// TIA Portal V17 export
// export: Created 2022-07-06T14:39:44.2676002Z, ExportSetting WithDefaults, DisplayName Totally Integrated Automation Portal, DisplayVersion V17 Update 4, DisplayName TIA Portal Openness, DisplayVersion V17 Update 4, DisplayName TIA Portal Version Control Interface, DisplayVersion V17, DisplayName STEP 7 Professional, DisplayVersion V17 Update 4, DisplayName STEP 7 CFC, DisplayVersion V17, DisplayName STEP 7 Safety, DisplayVersion V17, DisplayName WinCC Advanced, DisplayVersion V17 Update 4
DATA_BLOCK "HDB_STR"   // DB4300
{ S7_Optimized_Access := 'FALSE' }
NAME : DEV
VERSION : 0.1
// stored: AutoNumber false, DBAccessibleFromOPCUA true, IsOnlyStoredInLoadMemory false, IsWriteProtectedInAS false
   VAR RETAIN
      Cmd_ResetOsKnf1Top : Bool := FALSE;   // Knife 1 ss reset mileage
      Cmd_ResetOsKnf1Bot : Bool := FALSE;   // Knife 2 ss reset mileage
      Cmd_ResetOsSchp1 : Bool := FALSE;   // Knife 1 bs reset mileage
      Cmd_ResetOsKnf2Top : Bool := FALSE;   // Knife 1 ss reset mileage
      Cmd_ResetOsKnf2Bot : Bool := FALSE;   // Knife 2 ss reset mileage
      Cmd_ResetOsSchp2 : Bool := FALSE;   // Knife 1 bs reset mileage
      Cmd_ResetDsKnf1Top : Bool := FALSE;   // Knife 1 ss reset mileage
      Cmd_ResetDsKnf1Bot : Bool := FALSE;   // Knife 2 ss reset mileage
      Cmd_ResetDsSchp1 : Bool := FALSE;   // Knife 1 bs reset mileage
      Cmd_ResetDsKnf2Top : Bool := FALSE;   // Knife 1 ss reset mileage
      Cmd_ResetDsKnf2Bot : Bool := FALSE;   // Knife 2 ss reset mileage
      Cmd_ResetDsSchp2 : Bool := FALSE;   // Knife 1 bs reset mileage
      Cmd_FrcNotchInPos : Bool := FALSE;   // Notch in position
      Cmd_AutoRestart : Bool := FALSE;   // Line automatic start
      Cmd_StopRqst : Bool := FALSE;   // Line stop request
      Cmd_KnifeChngOsKnf1 : Bool := FALSE;   // Knife change operator Side Knife 1 request / Knife change BAL Side Knife 1 request
      Cmd_KnifeChngOsKnf2 : Bool := FALSE;   // Knife change operator Side Knife 2 request / Knife change BAL Side Knife 2 request
      Cmd_KnifeChngDsKnf1 : Bool := FALSE;   // Knife change drive Side Knife 1 request / Knife change Street Side Knife 1 request
      Cmd_KnifeChngDsKnf2 : Bool := FALSE;   // Knife change drive Side Knife 2 request / Knife change Street Side Knife 2 request
      Cmd_Spare23 { ExternalAccessible := 'False'; ExternalVisible := 'False'; ExternalWritable := 'False'} : Bool;
      Cmd_Spare24 { ExternalAccessible := 'False'; ExternalVisible := 'False'; ExternalWritable := 'False'} : Bool;
      Cmd_Spare25 { ExternalAccessible := 'False'; ExternalVisible := 'False'; ExternalWritable := 'False'} : Bool;
      Cmd_Spare26 { ExternalAccessible := 'False'; ExternalVisible := 'False'; ExternalWritable := 'False'} : Bool;
      Cmd_Spare27 { ExternalAccessible := 'False'; ExternalVisible := 'False'; ExternalWritable := 'False'} : Bool;
      Cmd_Spare31 { ExternalAccessible := 'False'; ExternalVisible := 'False'; ExternalWritable := 'False'} : Bool;
      Cmd_Spare32 { ExternalAccessible := 'False'; ExternalVisible := 'False'; ExternalWritable := 'False'} : Bool;
      Cmd_Spare33 { ExternalAccessible := 'False'; ExternalVisible := 'False'; ExternalWritable := 'False'} : Bool;
      Cmd_Spare34 { ExternalAccessible := 'False'; ExternalVisible := 'False'; ExternalWritable := 'False'} : Bool;
      Cmd_Spare35 { ExternalAccessible := 'False'; ExternalVisible := 'False'; ExternalWritable := 'False'} : Bool;
      Cmd_Spare36 { ExternalAccessible := 'False'; ExternalVisible := 'False'; ExternalWritable := 'False'} : Bool;
      Cmd_Spare37 { ExternalAccessible := 'False'; ExternalVisible := 'False'; ExternalWritable := 'False'} : Bool;
      Stat_NotchInPos : DInt := 4;   // Status notch in position
      Stat_AutoRestart : DInt := 6;   // Status Line automatic start
      Stat_StopRqst : DInt := 4;   // Status Line stop request
      Stat_KnifeChngOsKnf1 : DInt := 4;   // Status Knife change operator side Knife 1 request / Status Knife change BAL side Knife 1 request
      Stat_KnifeChngOsKnf2 : DInt := 1;   // Status Knife change operator side Knife 2 request / Status Knife change BAL side Knife 2 request
      Stat_KnifeChngDsKnf1 : DInt := 1;   // Status Knife change drive side Knife 1 request / Status Knife change Street side Knife 1 request
      Stat_KnifeChngDsKnf2 : DInt := 4;   // Status Knife change drive side Knife 2 request / Status Knife change Street side Knife 2 request
      Stat_Spare1 { ExternalAccessible := 'False'; ExternalVisible := 'False'; ExternalWritable := 'False'} : DInt;
      Stat_Spare2 { ExternalAccessible := 'False'; ExternalVisible := 'False'; ExternalWritable := 'False'} : DInt;
      Stat_Spare3 { ExternalAccessible := 'False'; ExternalVisible := 'False'; ExternalWritable := 'False'} : DInt;
      Stat_Spare4 { ExternalAccessible := 'False'; ExternalVisible := 'False'; ExternalWritable := 'False'} : DInt;
      Stat_Spare5 { ExternalAccessible := 'False'; ExternalVisible := 'False'; ExternalWritable := 'False'} : DInt;
      Chopper_Overspeed { S7_SetPoint := 'True'} : Real := 1.0;   // Chopper overspeed [%]
      MileageOsKnf1Top { S7_SetPoint := 'True'} : Real := 29.0;   // Mileage of knife 1 top OS / Mileage of knife 1 top Ss
      MileageOsKnf1Bot { S7_SetPoint := 'True'} : Real;   // Mileage of knife 1 bottom OS
      MileageOsSchp1 { S7_SetPoint := 'True'} : Real := 29.54701;   // Mileage of scrap chopper knife 1 OS / Mileage of scrap chopper knife 1 Ss
      MileageOsKnf2Top { S7_SetPoint := 'True'} : Real := 29.54701;   // Mileage of knife 2 top OS / Mileage of knife 1 top Ss
      MileageOsKnf2Bot { S7_SetPoint := 'True'} : Real;   // Mileage of knife 2 bottom OS
      MileageOsSchp2 { S7_SetPoint := 'True'} : Real := 18.93003;   // Mileage of scrap chopper knife 2 OS / Mileage of scrap chopper knife 2 Ss
      MileageDsKnf1Top { S7_SetPoint := 'True'} : Real := 29.54701;   // Mileage of knife 1 top DS / Mileage of knife 1 top Ss
      MileageDsKnf1Bot { S7_SetPoint := 'True'} : Real;   // Mileage of knife 1 bottom DS
      MileageDsSchp1 { S7_SetPoint := 'True'} : Real := 29.54701;   // Mileage of scrap chopper knife 1 DS / Mileage of scrap chopper knife 1 Ss
      MileageDsKnf2Top { S7_SetPoint := 'True'} : Real := 29.54701;   // Mileage of knife 2 top DS / Mileage of knife 1 top Ss
      MileageDsKnf2Bot { S7_SetPoint := 'True'} : Real;   // Mileage of knife 2 bottom DS
      MileageDsSchp2 { S7_SetPoint := 'True'} : Real := 18.93003;   // Mileage of scrap chopper knife 2 DS / Mileage of scrap chopper knife 2 Ss
      SetpOsGapKnf1 { S7_SetPoint := 'True'} : "SplSetpCtrl";   // Setpoint OS gap knife 1
      SetpOsOvlKnf1 { S7_SetPoint := 'True'} : "SplSetpCtrl";   // Setpoint OS overlap knife 1
      SetpOsSchp1 { S7_SetPoint := 'True'} : "SplSetpCtrl";   // Setpoint OS gap scrap chopper 1
      SetpOsGapKnf2 { S7_SetPoint := 'True'} : "SplSetpCtrl";   // Setpoint OS gap knife 2
      SetpOsOvlKnf2 { S7_SetPoint := 'True'} : "SplSetpCtrl";   // Setpoint OS overlap knife 2
      SetpOsSchp2 { S7_SetPoint := 'True'} : "SplSetpCtrl";   // Setpoint OS gap scrap chopper 2
      SetpDsGapKnf1 { S7_SetPoint := 'True'} : "SplSetpCtrl";   // Setpoint DS gap knife 1
      SetpDsOvlKnf1 { S7_SetPoint := 'True'} : "SplSetpCtrl";   // Setpoint DS overlap knife 1
      SetpDsSchp1 { S7_SetPoint := 'True'} : "SplSetpCtrl";   // Setpoint DS gap scrap chopper 1
      SetpDsGapKnf2 { S7_SetPoint := 'True'} : "SplSetpCtrl";   // Setpoint DS gap knife 2
      SetpDsOvlKnf2 { S7_SetPoint := 'True'} : "SplSetpCtrl";   // Setpoint DS overlap knife 2
      SetpDsSchp2 { S7_SetPoint := 'True'} : "SplSetpCtrl";   // Setpoint DS gap scrap chopper 2
      SetpTromWd { S7_SetPoint := 'True'} : "SplSetpCtrl";
   END_VAR
BEGIN
END_DATA_BLOCK
